TYPE Sapphire488LaserConfig EXTENDS DeviceConfiguration :
STRUCT
	SerialCommunication : SerialCommunication;
END_STRUCT
END_TYPE

(* stored: Version 1.1.0.1, ProductVersion 3.1.4024.12
   DUT Sapphire488LaserConfig: Id {2212f23b-f712-422c-9c29-d4a0741865a7} *)
